TEXTLIST EL1809_M_1
  1 = 'Fast Scan Origin' | chinese: 'Fast Scan 原点' | Chinese: 'Fast Scan 原点'
  2 = 'SpitUnit Origin' | chinese: '闪喷糟原点' | Chinese: '闪喷糟原点'
  3 = 'SpitUnit LimitP' | chinese: '闪喷糟极限' | Chinese: '闪喷糟极限'
  4 = 'Upper limit S1' | chinese: '压辊S1上限位' | Chinese: '压辊S1上限位'
  5 = 'Upper limit S2' | chinese: '压辊S2上限位' | Chinese: '压辊S2上限位'
  6 = 'Upper limit S3' | chinese: '压辊S3上限位' | Chinese: '压辊S3上限位'
  7 = 'Upper limit S4' | chinese: '压辊S4上限位' | Chinese: '压辊S4上限位'
  8 = 'Upper limit S5' | chinese: '压辊S5上限位' | Chinese: '压辊S5上限位'
  9 = 'Upper limit S6' | chinese: '压辊S6上限位' | Chinese: '压辊S6上限位'
  10 = 'Lower limit S1_1 ' | chinese: '压辊S1下限位1' | Chinese: '压辊S1下限位1'
  11 = 'Lower limit S1_2 ' | chinese: '压辊S1下限位2' | Chinese: '压辊S1下限位2'
  12 = 'Lower limit S1_3 ' | chinese: '压辊S1下限位3' | Chinese: '压辊S1下限位3'
  13 = 'Lower limit S1_4 ' | chinese: '压辊S1下限位4' | Chinese: '压辊S1下限位4'
  14 = 'Lower limit S1_5 ' | chinese: '压辊S1下限位5' | Chinese: '压辊S1下限位5'
  15 = 'Lower limit S1_6 ' | chinese: '压辊S1下限位6' | Chinese: '压辊S1下限位6'
  16 = 'Lower limit S1_7 ' | chinese: '压辊S1下限位7' | Chinese: '压辊S1下限位7'
   = ''
END_TEXTLIST

(* stored: Version 1.1.0.1, ProductVersion 3.1.4024.11
   TextList EL1809_M_1: Id {72810ef9-237b-48bb-983a-d3533e5d7315} *)
